// TIA Portal project "acacapdpd" (V16)

(* hardware
DEVICE "S71500/ET200MP station_1"  S7-1500 station
   slot 0: "Rail_0"  Rack  6ES7 590-1***0-0AA0
   slot 1: "PLC_1"  CPU 1512C-1 PN  6ES7 512-1CK01-0AB0  V2.8
      slot 3: "CPU display_1"  6ES7591-1AA00-0AA0
      slot 32768: "PROFINET interface_1"  X1
         slot 32769: "Port_1"  X1 P1
         slot 32770: "Port_2"  X1 P2
      slot 34817: "Virtual CP interface port_1"  Virtual CP interface port  Virtual CP interface port
DEVICE "HMI_1"  TP700 Comfort
   slot 0: "HMI_1"  TP700 Comfort  6AV2 124-0GC01-0AX0  16.0.0.0
   slot 1: "HMI_RT_1"  TP700 Comfort  6AV2 124-0GC01-0AX0  16.0.0.0
   slot 5: "HMI_1.IE_CP_1"  PROFINET Interface  16.0.0.0
      slot 1: "PROFINET Interface_1"  PROFINET Interface
         slot 1: "Port_1"  Port
         slot 2: "Port_2"  Port
   slot 7: "HMI_1.MPI/DP_CP_1"  MPI/DP Interface  16.0.0.0
*)

// ===== PLC "PLC_1"  CPU 1512C-1 PN =====

VAR_GLOBAL   // PLC tag table "Default tag table"
   "Mag" AT %I0.0 : Bool;
   "Slide 2" AT %I0.2 : Bool;
   "Slide 1" AT %I0.3 : Bool;
   "G is up" AT %I0.4 : Bool;
   "G is down" AT %I0.5 : Bool;
   "wp in mag pos" AT %I0.6 : Bool;
   "wp not black" AT %I0.7 : Bool;
   "Left" AT %Q0.2 : Bool;
   "Right" AT %Q0.0 : Bool;
   "Open G" AT %Q0.5 : Bool;
   "move G down" AT %Q0.7 : Bool;
   "Mag slide retracted" AT %I1.0 : Bool;
   "Mag slide advanced" AT %I1.2 : Bool;
   "EA push wp" AT %Q1.0 : Bool;
   "Red" AT %Q1.3 : Bool;
   "Green" AT %Q1.5 : Bool;
   "Yellow" AT %Q1.7 : Bool;
   "Clock_Byte" AT %MB20 : Byte;
   "Clock_10Hz" AT %M20.0 : Bool;
   "Clock_5Hz" AT %M20.1 : Bool;
   "Clock_2.5Hz" AT %M20.2 : Bool;
   "Clock_2Hz" AT %M20.3 : Bool;
   "Clock_1.25Hz" AT %M20.4 : Bool;
   "Clock_1Hz" AT %M20.5 : Bool;
   "Clock_0.625Hz" AT %M20.6 : Bool;
   "Clock_0.5Hz" AT %M20.7 : Bool;
   "Start" AT %M10.0 : Bool;
   "Reset" AT %M10.1 : Bool;
   "Stop" AT %M10.2 : Bool;
   "l_start" AT %M10.3 : Bool;
   "l_reset" AT %M10.4 : Bool;
   "l_Q1" AT %M10.5 : Bool;
   "l_Q2" AT %M10.6 : Bool;
   "Key" AT %M10.7 : Bool;
   "step" AT %MW0 : Int;
END_VAR

ORGANIZATION_BLOCK "Main"   // OB1, FBD, ProgramCycle
TITLE = "Main Program Sweep (Cycle)"
{ S7_Optimized_Access := 'TRUE' }
VERSION : 0.1
   VAR_INPUT
      Initial_Call : Bool;   // Initial call of this OB
      Remanence : Bool;   // =True, if remanent data are available
   END_VAR
   VAR_TEMP   // added for the SCL form of the ladder/FBD networks
      _w1 : Bool;
   END_VAR
BEGIN

REGION Network 1
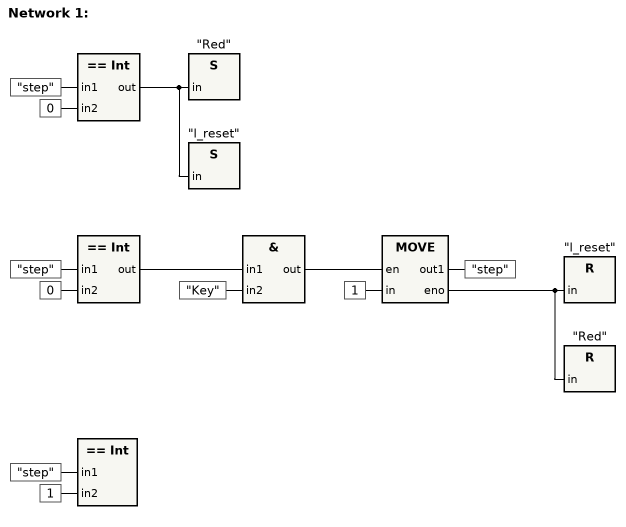
   IF "step" = 0 THEN
       "Red" := TRUE;
       "l_reset" := TRUE;
   END_IF;
   #_w1 := ("step" = 0) AND "Key";
   IF #_w1 THEN
       "step" := 1;
       "l_reset" := FALSE;
       "Red" := FALSE;
   END_IF;
END_REGION
END_ORGANIZATION_BLOCK

(* ===== HMI "HMI_RT_1" =====
connection "HMI_Connection_1": ETHERNET, S7_1500_OMS

HMI tags "Default tag table"
   "Start" : Bool = PLC Start AT %M10.0, 100 ms
   "Stop" : Bool = PLC Stop AT %M10.2, 100 ms
   "Reset" : Bool = PLC Reset AT %M10.1, 100 ms
   "l_start" : Bool = PLC l_start AT %M10.3, 100 ms
   "l_reset" : Bool = PLC l_reset AT %M10.4, 100 ms
   "l_Q1" : Bool = PLC l_Q1 AT %M10.5, 100 ms
   "l_Q2" : Bool = PLC l_Q2 AT %M10.6, 100 ms
   "Key" : Bool = PLC Key AT %M10.7, 100 ms
*)